KUKA KRL program: probetasprueba.src, probetasprueba.dat

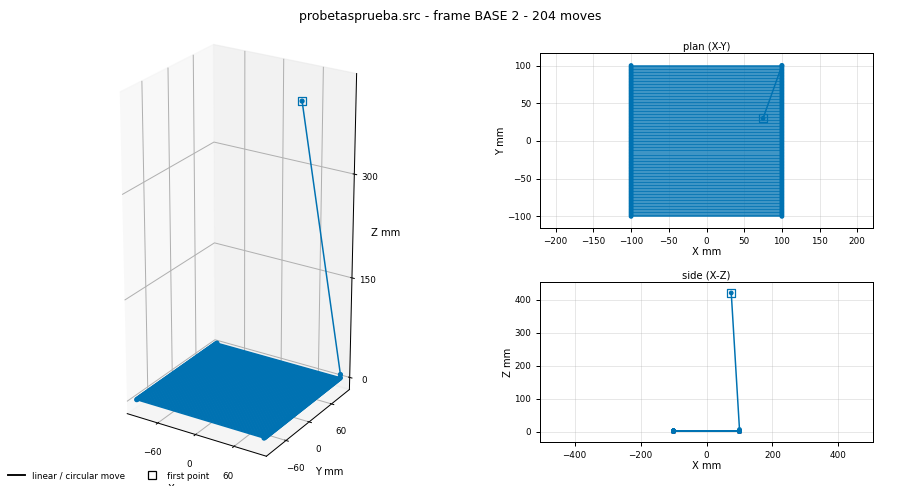
[picture p0: tool path of probetasprueba.src in frame BASE 2, 204 of 206 moves have a stored position in this frame; points joined in program order, loops and branches not executed]
--- probetasprueba.src ---
&ACCESS RVP
&PARAM TEMPLATE = C:\KRC\Roboter\Template\vorgabe
&PARAM EDITMASK = *
DEF probetasprueba( )
;FOLD INI;%{PE}%V3.2.0,%MKUKATPBASIS,%CINIT,%VCOMMON,%P
;FOLD BAS INI;%{E}%V3.2.0,%MKUKATPBASIS,%CINIT,%VINIT,%P
GLOBAL INTERRUPT DECL 3 WHEN $STOPMESS==TRUE DO IR_STOPM ( )
INTERRUPT ON 3
BAS (#INITMOV,0 )
;ENDFOLD (BAS INI)
;FOLD A20 INI;%{E}%V3.2.0,%MKUKATPA20,%CINIT,%VINIT,%P
IF ARC20==TRUE THEN
A20 (ARC_INI)
INTERRUPT DECL 6 WHEN $CYCFLAG[3]==FALSE DO A20(TECH_STOP2)
ENDIF
;ENDFOLD (A20 INI)
;FOLD A10 INI;%{E}%V3.2.0,%MKUKATPARC,%CINIT,%VINIT,%P
IF A10_OPTION==#ACTIVE THEN
INTERRUPT DECL 4 WHEN $CYCFLAG[2]==FALSE DO A10 (#APPL_ERROR)
INTERRUPT DECL 7 WHEN A_ARC_SWI==#ACTIVE DO A10 (#ARC_SEAM)
INTERRUPT DECL 5 WHEN A_FLY_ARC==TRUE DO A10 (#HPU_ARC)
INTERRUPT  ON 5
A10_INI ( )
ENDIF
;ENDFOLD (A10 INI)
;FOLD GRIPPER INI;%{E}%V3.2.0,%MKUKATPGRIPPER,%CINIT,%VINIT,%P
USER_GRP(0,DUMMY,DUMMY,GDEFAULT)
;ENDFOLD (GRIPPER INI)
;FOLD SPOT INI;%{E}%V3.2.0,%MKUKATPSPOT,%CINIT,%VINIT,%P
USERSPOT(#INIT)
;ENDFOLD (SPOT INI)
;FOLD TOUCHSENSE INI;%{E}%V3.2.0,%MKUKATPTS,%CINIT,%VINIT,%P
IF H70_OPTION THEN
INTERRUPT DECL 15 WHEN $MEAS_PULSE[TOUCH_I[TOUCH_ACTIVE].IN_NR] DO H70 (6,CD0 )
INTERRUPT DECL 16 WHEN $ZERO_MOVE DO H70 (7,CD0 )
INTERRUPT DECL 17 WHEN $TECHPAR_C[FG_TOUCH,8]>0.5 DO H70 (8,CD0)
H70 (1,CD0 )
ENDIF
;ENDFOLD (TOUCHSENSE INI)
;FOLD USER INI;%{E}%V3.2.0,%MKUKATPUSER,%CINIT,%VINIT,%P
;Make your modifications here
;ENDFOLD (USER INI)
;ENDFOLD (INI)
; SPEED PTP FOR AXIS
$VEL_AXIS[1] = 15
$VEL_AXIS[2] = 15
$VEL_AXIS[3] = 15
$VEL_AXIS[4] = 15
$VEL_AXIS[5] = 15
$VEL_AXIS[6] = 15
;SMOOTHNESS
$APO.CDIS = 2
;ADVANCE
$ADVANCE = 3
;SET TOOL AND BASE
$TOOL = TOOL_DATA[3]
$BASE = BASE_DATA[2]
;HOME
;FOLD PTP HOME Vel=10% DEFAULT
$BWDSTART=FALSE
$H_POS=XHOME
PDAT_ACT=PDEFAULT
FDAT_ACT=FHOME
BAS(#PTP_DAT )
BAS (#VEL_PTP,10 )
PTP XHOME
;ENDFOLD
;USER PROGRAM
;SPEED $VEL.CP
$VEL.CP=0.05
; OUT[TEMP] = 200
; OUT[vent] = 1
; OUT[RPM] = 50
; USER POSES CALLS
PTP {X 75, Y 30, Z 420, A 0, B 90, C 0}
; USER POSES CALLS
LIN {X 100.0, Y 100.0, Z 6, A 0, B 90, C 0} C_DIS
WAIT SEC 1
$OUT[1] = TRUE
LIN {X 100.0, Y 100.0, Z 1, A 0, B 90, C 0} C_DIS
LIN {X -100.0, Y 100.0, Z 1, A 0, B 90, C 0} C_DIS
LIN {X -100.0, Y 98.0, Z 1, A 0, B 90, C 0} C_DIS
LIN {X 100.0, Y 98.0, Z 1, A 0, B 90, C 0} C_DIS
LIN {X 100.0, Y 96.0, Z 1, A 0, B 90, C 0} C_DIS
LIN {X -100.0, Y 96.0, Z 1, A 0, B 90, C 0} C_DIS
LIN {X -100.0, Y 94.0, Z 1, A 0, B 90, C 0} C_DIS
LIN {X 100.0, Y 94.0, Z 1, A 0, B 90, C 0} C_DIS
LIN {X 100.0, Y 92.0, Z 1, A 0, B 90, C 0} C_DIS
LIN {X -100.0, Y 92.0, Z 1, A 0, B 90, C 0} C_DIS
LIN {X -100.0, Y 90.0, Z 1, A 0, B 90, C 0} C_DIS
LIN {X 100.0, Y 90.0, Z 1, A 0, B 90, C 0} C_DIS
LIN {X 100.0, Y 88.0, Z 1, A 0, B 90, C 0} C_DIS
LIN {X -100.0, Y 88.0, Z 1, A 0, B 90, C 0} C_DIS
LIN {X -100.0, Y 86.0, Z 1, A 0, B 90, C 0} C_DIS
LIN {X 100.0, Y 86.0, Z 1, A 0, B 90, C 0} C_DIS
LIN {X 100.0, Y 84.0, Z 1, A 0, B 90, C 0} C_DIS
LIN {X -100.0, Y 84.0, Z 1, A 0, B 90, C 0} C_DIS
LIN {X -100.0, Y 82.0, Z 1, A 0, B 90, C 0} C_DIS
LIN {X 100.0, Y 82.0, Z 1, A 0, B 90, C 0} C_DIS
LIN {X 100.0, Y 80.0, Z 1, A 0, B 90, C 0} C_DIS
LIN {X -100.0, Y 80.0, Z 1, A 0, B 90, C 0} C_DIS
LIN {X -100.0, Y 78.0, Z 1, A 0, B 90, C 0} C_DIS
LIN {X 100.0, Y 78.0, Z 1, A 0, B 90, C 0} C_DIS
LIN {X 100.0, Y 76.0, Z 1, A 0, B 90, C 0} C_DIS
LIN {X -100.0, Y 76.0, Z 1, A 0, B 90, C 0} C_DIS
LIN {X -100.0, Y 74.0, Z 1, A 0, B 90, C 0} C_DIS
LIN {X 100.0, Y 74.0, Z 1, A 0, B 90, C 0} C_DIS
LIN {X 100.0, Y 72.0, Z 1, A 0, B 90, C 0} C_DIS
LIN {X -100.0, Y 72.0, Z 1, A 0, B 90, C 0} C_DIS
LIN {X -100.0, Y 70.0, Z 1, A 0, B 90, C 0} C_DIS
LIN {X 100.0, Y 70.0, Z 1, A 0, B 90, C 0} C_DIS
LIN {X 100.0, Y 68.0, Z 1, A 0, B 90, C 0} C_DIS
LIN {X -100.0, Y 68.0, Z 1, A 0, B 90, C 0} C_DIS
LIN {X -100.0, Y 66.0, Z 1, A 0, B 90, C 0} C_DIS
LIN {X 100.0, Y 66.0, Z 1, A 0, B 90, C 0} C_DIS
LIN {X 100.0, Y 64.0, Z 1, A 0, B 90, C 0} C_DIS
LIN {X -100.0, Y 64.0, Z 1, A 0, B 90, C 0} C_DIS
LIN {X -100.0, Y 62.0, Z 1, A 0, B 90, C 0} C_DIS
LIN {X 100.0, Y 62.0, Z 1, A 0, B 90, C 0} C_DIS
LIN {X 100.0, Y 60.0, Z 1, A 0, B 90, C 0} C_DIS
LIN {X -100.0, Y 60.0, Z 1, A 0, B 90, C 0} C_DIS
LIN {X -100.0, Y 58.0, Z 1, A 0, B 90, C 0} C_DIS
LIN {X 100.0, Y 58.0, Z 1, A 0, B 90, C 0} C_DIS
LIN {X 100.0, Y 56.0, Z 1, A 0, B 90, C 0} C_DIS
LIN {X -100.0, Y 56.0, Z 1, A 0, B 90, C 0} C_DIS
LIN {X -100.0, Y 54.0, Z 1, A 0, B 90, C 0} C_DIS
LIN {X 100.0, Y 54.0, Z 1, A 0, B 90, C 0} C_DIS
LIN {X 100.0, Y 52.0, Z 1, A 0, B 90, C 0} C_DIS
LIN {X -100.0, Y 52.0, Z 1, A 0, B 90, C 0} C_DIS
LIN {X -100.0, Y 50.0, Z 1, A 0, B 90, C 0} C_DIS
LIN {X 100.0, Y 50.0, Z 1, A 0, B 90, C 0} C_DIS
LIN {X 100.0, Y 48.0, Z 1, A 0, B 90, C 0} C_DIS
LIN {X -100.0, Y 48.0, Z 1, A 0, B 90, C 0} C_DIS
LIN {X -100.0, Y 46.0, Z 1, A 0, B 90, C 0} C_DIS
LIN {X 100.0, Y 46.0, Z 1, A 0, B 90, C 0} C_DIS
LIN {X 100.0, Y 44.0, Z 1, A 0, B 90, C 0} C_DIS
LIN {X -100.0, Y 44.0, Z 1, A 0, B 90, C 0} C_DIS
LIN {X -100.0, Y 42.0, Z 1, A 0, B 90, C 0} C_DIS
LIN {X 100.0, Y 42.0, Z 1, A 0, B 90, C 0} C_DIS
LIN {X 100.0, Y 40.0, Z 1, A 0, B 90, C 0} C_DIS
LIN {X -100.0, Y 40.0, Z 1, A 0, B 90, C 0} C_DIS
LIN {X -100.0, Y 38.0, Z 1, A 0, B 90, C 0} C_DIS
LIN {X 100.0, Y 38.0, Z 1, A 0, B 90, C 0} C_DIS
LIN {X 100.0, Y 36.0, Z 1, A 0, B 90, C 0} C_DIS
LIN {X -100.0, Y 36.0, Z 1, A 0, B 90, C 0} C_DIS
LIN {X -100.0, Y 34.0, Z 1, A 0, B 90, C 0} C_DIS
LIN {X 100.0, Y 34.0, Z 1, A 0, B 90, C 0} C_DIS
LIN {X 100.0, Y 32.0, Z 1, A 0, B 90, C 0} C_DIS
LIN {X -100.0, Y 32.0, Z 1, A 0, B 90, C 0} C_DIS
LIN {X -100.0, Y 30.0, Z 1, A 0, B 90, C 0} C_DIS
LIN {X 100.0, Y 30.0, Z 1, A 0, B 90, C 0} C_DIS
LIN {X 100.0, Y 28.0, Z 1, A 0, B 90, C 0} C_DIS
LIN {X -100.0, Y 28.0, Z 1, A 0, B 90, C 0} C_DIS
LIN {X -100.0, Y 26.0, Z 1, A 0, B 90, C 0} C_DIS
LIN {X 100.0, Y 26.0, Z 1, A 0, B 90, C 0} C_DIS
LIN {X 100.0, Y 24.0, Z 1, A 0, B 90, C 0} C_DIS
LIN {X -100.0, Y 24.0, Z 1, A 0, B 90, C 0} C_DIS
LIN {X -100.0, Y 22.0, Z 1, A 0, B 90, C 0} C_DIS
LIN {X 100.0, Y 22.0, Z 1, A 0, B 90, C 0} C_DIS
LIN {X 100.0, Y 20.0, Z 1, A 0, B 90, C 0} C_DIS
LIN {X -100.0, Y 20.0, Z 1, A 0, B 90, C 0} C_DIS
LIN {X -100.0, Y 18.0, Z 1, A 0, B 90, C 0} C_DIS
LIN {X 100.0, Y 18.0, Z 1, A 0, B 90, C 0} C_DIS
LIN {X 100.0, Y 16.0, Z 1, A 0, B 90, C 0} C_DIS
LIN {X -100.0, Y 16.0, Z 1, A 0, B 90, C 0} C_DIS
LIN {X -100.0, Y 14.0, Z 1, A 0, B 90, C 0} C_DIS
LIN {X 100.0, Y 14.0, Z 1, A 0, B 90, C 0} C_DIS
LIN {X 100.0, Y 12.0, Z 1, A 0, B 90, C 0} C_DIS
LIN {X -100.0, Y 12.0, Z 1, A 0, B 90, C 0} C_DIS
LIN {X -100.0, Y 10.0, Z 1, A 0, B 90, C 0} C_DIS
LIN {X 100.0, Y 10.0, Z 1, A 0, B 90, C 0} C_DIS
LIN {X 100.0, Y 8.0, Z 1, A 0, B 90, C 0} C_DIS
LIN {X -100.0, Y 8.0, Z 1, A 0, B 90, C 0} C_DIS
LIN {X -100.0, Y 6.0, Z 1, A 0, B 90, C 0} C_DIS
LIN {X 100.0, Y 6.0, Z 1, A 0, B 90, C 0} C_DIS
LIN {X 100.0, Y 4.0, Z 1, A 0, B 90, C 0} C_DIS
LIN {X -100.0, Y 4.0, Z 1, A 0, B 90, C 0} C_DIS
LIN {X -100.0, Y 2.0, Z 1, A 0, B 90, C 0} C_DIS
LIN {X 100.0, Y 2.0, Z 1, A 0, B 90, C 0} C_DIS
LIN {X 100.0, Y 0.0, Z 1, A 0, B 90, C 0} C_DIS
LIN {X -100.0, Y 0.0, Z 1, A 0, B 90, C 0} C_DIS
LIN {X -100.0, Y -2.0, Z 1, A 0, B 90, C 0} C_DIS
LIN {X 100.0, Y -2.0, Z 1, A 0, B 90, C 0} C_DIS
LIN {X 100.0, Y -4.0, Z 1, A 0, B 90, C 0} C_DIS
LIN {X -100.0, Y -4.0, Z 1, A 0, B 90, C 0} C_DIS
LIN {X -100.0, Y -6.0, Z 1, A 0, B 90, C 0} C_DIS
LIN {X 100.0, Y -6.0, Z 1, A 0, B 90, C 0} C_DIS
LIN {X 100.0, Y -8.0, Z 1, A 0, B 90, C 0} C_DIS
LIN {X -100.0, Y -8.0, Z 1, A 0, B 90, C 0} C_DIS
LIN {X -100.0, Y -10.0, Z 1, A 0, B 90, C 0} C_DIS
LIN {X 100.0, Y -10.0, Z 1, A 0, B 90, C 0} C_DIS
LIN {X 100.0, Y -12.0, Z 1, A 0, B 90, C 0} C_DIS
LIN {X -100.0, Y -12.0, Z 1, A 0, B 90, C 0} C_DIS
LIN {X -100.0, Y -14.0, Z 1, A 0, B 90, C 0} C_DIS
LIN {X 100.0, Y -14.0, Z 1, A 0, B 90, C 0} C_DIS
LIN {X 100.0, Y -16.0, Z 1, A 0, B 90, C 0} C_DIS
LIN {X -100.0, Y -16.0, Z 1, A 0, B 90, C 0} C_DIS
LIN {X -100.0, Y -18.0, Z 1, A 0, B 90, C 0} C_DIS
LIN {X 100.0, Y -18.0, Z 1, A 0, B 90, C 0} C_DIS
LIN {X 100.0, Y -20.0, Z 1, A 0, B 90, C 0} C_DIS
LIN {X -100.0, Y -20.0, Z 1, A 0, B 90, C 0} C_DIS
LIN {X -100.0, Y -22.0, Z 1, A 0, B 90, C 0} C_DIS
LIN {X 100.0, Y -22.0, Z 1, A 0, B 90, C 0} C_DIS
LIN {X 100.0, Y -24.0, Z 1, A 0, B 90, C 0} C_DIS
LIN {X -100.0, Y -24.0, Z 1, A 0, B 90, C 0} C_DIS
LIN {X -100.0, Y -26.0, Z 1, A 0, B 90, C 0} C_DIS
LIN {X 100.0, Y -26.0, Z 1, A 0, B 90, C 0} C_DIS
LIN {X 100.0, Y -28.0, Z 1, A 0, B 90, C 0} C_DIS
LIN {X -100.0, Y -28.0, Z 1, A 0, B 90, C 0} C_DIS
LIN {X -100.0, Y -30.0, Z 1, A 0, B 90, C 0} C_DIS
LIN {X 100.0, Y -30.0, Z 1, A 0, B 90, C 0} C_DIS
LIN {X 100.0, Y -32.0, Z 1, A 0, B 90, C 0} C_DIS
LIN {X -100.0, Y -32.0, Z 1, A 0, B 90, C 0} C_DIS
LIN {X -100.0, Y -34.0, Z 1, A 0, B 90, C 0} C_DIS
LIN {X 100.0, Y -34.0, Z 1, A 0, B 90, C 0} C_DIS
LIN {X 100.0, Y -36.0, Z 1, A 0, B 90, C 0} C_DIS
LIN {X -100.0, Y -36.0, Z 1, A 0, B 90, C 0} C_DIS
LIN {X -100.0, Y -38.0, Z 1, A 0, B 90, C 0} C_DIS
LIN {X 100.0, Y -38.0, Z 1, A 0, B 90, C 0} C_DIS
LIN {X 100.0, Y -40.0, Z 1, A 0, B 90, C 0} C_DIS
LIN {X -100.0, Y -40.0, Z 1, A 0, B 90, C 0} C_DIS
LIN {X -100.0, Y -42.0, Z 1, A 0, B 90, C 0} C_DIS
LIN {X 100.0, Y -42.0, Z 1, A 0, B 90, C 0} C_DIS
LIN {X 100.0, Y -44.0, Z 1, A 0, B 90, C 0} C_DIS
LIN {X -100.0, Y -44.0, Z 1, A 0, B 90, C 0} C_DIS
LIN {X -100.0, Y -46.0, Z 1, A 0, B 90, C 0} C_DIS
LIN {X 100.0, Y -46.0, Z 1, A 0, B 90, C 0} C_DIS
LIN {X 100.0, Y -48.0, Z 1, A 0, B 90, C 0} C_DIS
LIN {X -100.0, Y -48.0, Z 1, A 0, B 90, C 0} C_DIS
LIN {X -100.0, Y -50.0, Z 1, A 0, B 90, C 0} C_DIS
LIN {X 100.0, Y -50.0, Z 1, A 0, B 90, C 0} C_DIS
LIN {X 100.0, Y -52.0, Z 1, A 0, B 90, C 0} C_DIS
LIN {X -100.0, Y -52.0, Z 1, A 0, B 90, C 0} C_DIS
LIN {X -100.0, Y -54.0, Z 1, A 0, B 90, C 0} C_DIS
LIN {X 100.0, Y -54.0, Z 1, A 0, B 90, C 0} C_DIS
LIN {X 100.0, Y -56.0, Z 1, A 0, B 90, C 0} C_DIS
LIN {X -100.0, Y -56.0, Z 1, A 0, B 90, C 0} C_DIS
LIN {X -100.0, Y -58.0, Z 1, A 0, B 90, C 0} C_DIS
LIN {X 100.0, Y -58.0, Z 1, A 0, B 90, C 0} C_DIS
LIN {X 100.0, Y -60.0, Z 1, A 0, B 90, C 0} C_DIS
LIN {X -100.0, Y -60.0, Z 1, A 0, B 90, C 0} C_DIS
LIN {X -100.0, Y -62.0, Z 1, A 0, B 90, C 0} C_DIS
LIN {X 100.0, Y -62.0, Z 1, A 0, B 90, C 0} C_DIS
LIN {X 100.0, Y -64.0, Z 1, A 0, B 90, C 0} C_DIS
LIN {X -100.0, Y -64.0, Z 1, A 0, B 90, C 0} C_DIS
LIN {X -100.0, Y -66.0, Z 1, A 0, B 90, C 0} C_DIS
LIN {X 100.0, Y -66.0, Z 1, A 0, B 90, C 0} C_DIS
LIN {X 100.0, Y -68.0, Z 1, A 0, B 90, C 0} C_DIS
LIN {X -100.0, Y -68.0, Z 1, A 0, B 90, C 0} C_DIS
LIN {X -100.0, Y -70.0, Z 1, A 0, B 90, C 0} C_DIS
LIN {X 100.0, Y -70.0, Z 1, A 0, B 90, C 0} C_DIS
LIN {X 100.0, Y -72.0, Z 1, A 0, B 90, C 0} C_DIS
LIN {X -100.0, Y -72.0, Z 1, A 0, B 90, C 0} C_DIS
LIN {X -100.0, Y -74.0, Z 1, A 0, B 90, C 0} C_DIS
LIN {X 100.0, Y -74.0, Z 1, A 0, B 90, C 0} C_DIS
LIN {X 100.0, Y -76.0, Z 1, A 0, B 90, C 0} C_DIS
LIN {X -100.0, Y -76.0, Z 1, A 0, B 90, C 0} C_DIS
LIN {X -100.0, Y -78.0, Z 1, A 0, B 90, C 0} C_DIS
LIN {X 100.0, Y -78.0, Z 1, A 0, B 90, C 0} C_DIS
LIN {X 100.0, Y -80.0, Z 1, A 0, B 90, C 0} C_DIS
LIN {X -100.0, Y -80.0, Z 1, A 0, B 90, C 0} C_DIS
LIN {X -100.0, Y -82.0, Z 1, A 0, B 90, C 0} C_DIS
LIN {X 100.0, Y -82.0, Z 1, A 0, B 90, C 0} C_DIS
LIN {X 100.0, Y -84.0, Z 1, A 0, B 90, C 0} C_DIS
LIN {X -100.0, Y -84.0, Z 1, A 0, B 90, C 0} C_DIS
LIN {X -100.0, Y -86.0, Z 1, A 0, B 90, C 0} C_DIS
LIN {X 100.0, Y -86.0, Z 1, A 0, B 90, C 0} C_DIS
LIN {X 100.0, Y -88.0, Z 1, A 0, B 90, C 0} C_DIS
LIN {X -100.0, Y -88.0, Z 1, A 0, B 90, C 0} C_DIS
LIN {X -100.0, Y -90.0, Z 1, A 0, B 90, C 0} C_DIS
LIN {X 100.0, Y -90.0, Z 1, A 0, B 90, C 0} C_DIS
LIN {X 100.0, Y -92.0, Z 1, A 0, B 90, C 0} C_DIS
LIN {X -100.0, Y -92.0, Z 1, A 0, B 90, C 0} C_DIS
LIN {X -100.0, Y -94.0, Z 1, A 0, B 90, C 0} C_DIS
LIN {X 100.0, Y -94.0, Z 1, A 0, B 90, C 0} C_DIS
LIN {X 100.0, Y -96.0, Z 1, A 0, B 90, C 0} C_DIS
LIN {X -100.0, Y -96.0, Z 1, A 0, B 90, C 0} C_DIS
LIN {X -100.0, Y -98.0, Z 1, A 0, B 90, C 0} C_DIS
LIN {X 100.0, Y -98.0, Z 1, A 0, B 90, C 0} C_DIS
LIN {X 100.0, Y -100.0, Z 1, A 0, B 90, C 0} C_DIS
LIN {X -100.0, Y -100.0, Z 1, A 0, B 90, C 0} C_DIS
$OUT[1] = FALSE

;Wait for
; END POSITION FOR
;END USER CODE
;HOME
;FOLD PTP HOME Vel=10% DEFAULT
$BWDSTART=FALSE
$H_POS=XHOME
PDAT_ACT=PDEFAULT
FDAT_ACT=FHOME
BAS(#PTP_DAT )
BAS (#VEL_PTP,10 )
PTP XHOME
;ENDFOLD
END

--- probetasprueba.dat ---
DEFDAT probetasprueba()
ENDDAT
